FUNCTION_BLOCK FB_AX5000_ReadDiagCode
VAR_INPUT
	Cmd_ReadDiagCode						:	BOOL;
END_VAR
VAR_OUTPUT

	Sts_ActualDiagCode						:	UDINT;
	Sts_DiagList							:	Tc2_Drive.ST_SoE_DiagNumList;	
	Sts_Error								:	BOOL;
END_VAR
VAR

	// AX5000/SoE
	SoEReset 								:	Tc2_Mc2_Drive.FB_SoEReset;
	SoERead 								:	Tc2_Mc2_Drive.FB_SoERead;
	SoEReadValue 							:	UINT;
	ReadSOE_LIST 							:	Tc2_MC2_Drive.FB_SoEReadDiagNumberList;
	StepControl								:	UINT;

END_VAR
VAR_IN_OUT
	Axis									:	Tc2_mc2.AXIS_REF;
END_VAR

// AX5000 Read Diag Codes - With standard blocks
// This block is made for inspirational purposes.
// Please make your ovn version that complies with your / your company´s programming vision
// Version 1.0 - Initial Version
//-----------------------------------------------------------------------------------------

ReadSOE_LIST(Axis := Axis, Timeout := DEFAULT_ADS_TIMEOUT, pDiagNumber := ADR(Sts_DiagList),Size:= SIZEOF(Sts_DiagList));
SoERead(Axis:=Axis,Element:=16#40,pDstBuf:=ADR(SoEReadValue),BufLen:=SIZEOF(SoEReadValue));
SoEReset(Axis:=Axis);

CASE StepControl OF
	
	0:
		IF Cmd_ReadDiagCode THEN
			StepControl := 10;
		END_IF

	10: // Sercos Axis
	
		ReadSOE_LIST.Execute := TRUE;
		IF ReadSOE_LIST.Busy THEN
			StepControl :=20;
		END_IF
		IF ReadSOE_LIST.Error THEN
			Sts_Error :=1;
			StepControl :=666;
		END_IF
		
	20:
		IF NOT ReadSOE_LIST.Busy THEN
			Sts_ActualDiagCode := Sts_DiagList.arrDiagNumbers[Sts_DiagList.iActualSize];
			StepControl :=30;
		END_IF
		
		IF ReadSOE_LIST.Error THEN
			Sts_Error :=1;
			StepControl :=666;
		END_IF
		
	30:
		IF NOT Cmd_ReadDiagCode THEN
			StepControl :=0;
		END_IF
	
	
	666:
		IF NOT Cmd_ReadDiagCode THEN
			Sts_Error :=0;
			StepControl :=0;
		END_IF
		
END_CASE

END_FUNCTION_BLOCK

(* stored: Version 1.1.0.1, ProductVersion 3.1.4024.14
   POU FB_AX5000_ReadDiagCode: Id {8301114d-fc25-45be-b65b-7c58c49b2640}, SpecialFunc None *)
